Omron CX-Programmer project NewProject (CX-Programmer 9.70)

# PLC NewPLC1: CP1E E20

## Global symbols (name address type ; comment)
0.02 BOOL  ; start
0.03 BOOL  ; stop
100.00 BOOL  ; output

## Program NewProgram1 (cyclic task 0)

### Section Section1

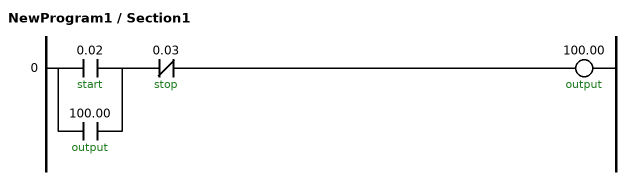
; rung 0
LD 0.02  ; start
OR 100.00  ; output
ANDNOT 0.03  ; stop
OUT 100.00  ; output

### Section END
; rung 0
END(001)